TYPE TcoDaqDataItemImplementation EXTENDS TcoCore.TcoDaqItem :
STRUCT
	Data : TcoDaqData; 
END_STRUCT
END_TYPE

(* stored: Version 1.1.0.1
   DUT TcoDaqDataItemImplementation: Id {e0905e98-2f17-0a1e-3144-14af9c8203d1} *)
